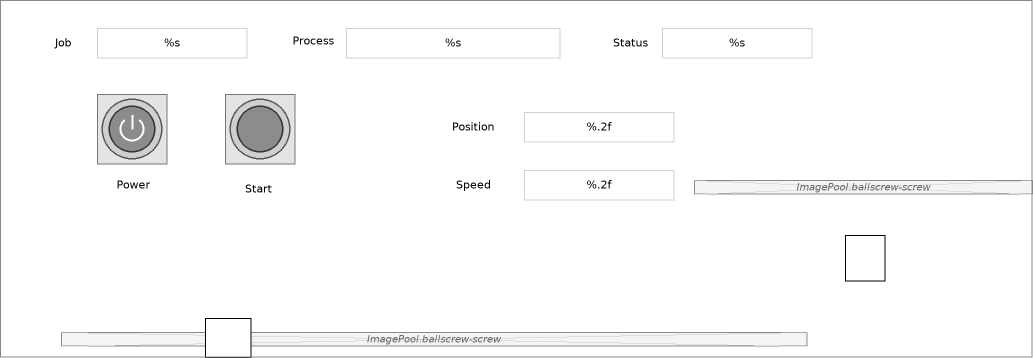
VISUALIZATION Visualization  // 1033x358
    PushSwitch (225,94 70x70), variable: demo3.bStart, behaviour: TOGGLE, style: Switch-PushSwitch-Gray
    Textfield (97,28 150x30), "%s", text variable: demo3.runner.job_event_cyclic_output.event_message.job_id
    Label (280,26 67x30), "Process"
    Label (30,28 67x30), "Job"
    PowerSwitch (97,94 70x70), variable: demo3.bPower, behaviour: TOGGLE, style: Switch-PowerSwitch-Gray
    Textfield (524,112 150x30), "%.2f", text variable: GVL.axis1.NcToPlc.ActPos
    Textfield (346,28 214x30), "%s", text variable: demo3.runner.job_event_cyclic_output.event_message.subject
    Textfield (662,28 150x30), "%s", text variable: demo3.runner.job_event_cyclic_output.event_message.new_state
    Label (597,28 67x30), "Status"
    Textfield (524,170 150x30), "%.2f", text variable: GVL.axis1.NcToPlc.ActVelo
    Image (61,332 746x14), image: ImagePool.ballscrew-screw
    Rectangle (205,318 46x40)
        p3560616238: GVL.axis1.NcToPlc.ActPos / 10.0
    Label (100,170 67x30), "Power"
    Label (225,174 67x30), "Start"
    Label (440,112 67x30), "Position"
    Label (440,170 67x30), "Speed"
    Image (694,180 339x14), angle 90, image: ImagePool.ballscrew-screw
    Rectangle (842,238 46x40), angle 270
        p2738717112: GVL.axis2.NcToPlc.ActPos / 10.0
END_VISUALIZATION

(* stored: Version 1.1.0.1, ProductVersion 3.1.4026.17
   Visu Visualization: Id {eb6f1f97-96f5-4efa-9e51-faa3758276d5} *)
